PROGRAM LOGPROCESS
VAR_INPUT
	spLogEvent	: STRING;
	spLogComp	: STRING;
	spLogAction	: STRING;
	spLogStatus	: STRING;
	plogFlag		: BOOL;
END_VAR
VAR_OUTPUT
	plog_complete : BOOL := FALSE;
	plog_error	 : BOOL := FALSE;
END_VAR
VAR
	fb_TimeStamp : FB_UpdateTimeStamp ();
	fbCreateDir	 : FB_CreateDir;
	fbFileOpen	 : FB_FileOpen;
	fbFileWrite	 : FB_FilePuts;
	fbFileClose	 : FB_FileClose;
	plog_state	 : ( INIT, 
					 CREATE_DIR, 
					 FILE_OPEN,
					 WRITE_TITLE,
					 WRITE_LOG, 
					 FILE_CLOSE,
					 CLEAR, 
					 ERROR);
					
	pwritepLog	 : STRING[255];
	pwriteTitle	 : STRING;
	spFolderName	 : STRING;
	spwFolderName	 : STRING;
	spFileName	 : STRING;
	spTextLog	 : STRING;
	spwTextLog	 : STRING;
	plastFileName : STRING;	
	spwLogEvent	: STRING;
	spwLogComp	: STRING;
	spwLogAction	: STRING;
	spwLogStatus	: STRING;
	
END_VAR

IF spLogComp<>spwLogComp OR spLogAction<>spwLogAction OR spLogStatus<>spwLogStatus THEN
//	spwLogEvent		:= spLogEvent;
	spwLogComp		:= spLogComp;
	spwLogAction	:= spLogAction;
	spwLogStatus	:= spLogStatus;
ELSE
	RETURN;
END_IF

spTextLog := str_concat(spwLogComp,spwLogAction,spwLogStatus);

WHILE plogFlag DO
	CASE plog_state OF
		// INIT -------------------------------------------------------------------
		INIT:
			plog_complete	:= FALSE;
			plog_error		:= FALSE;
			plog_state 		:= CREATE_DIR;
			fbCreateDir(bExecute:= FALSE);
	
		// CREATE_DIR -------------------------------------------------------------			
		CREATE_DIR:	
			spFolderName := CONCAT('C:\Users\Administrator\Desktop\log\PROCESS\', MAIN.fb_TimeStamp.SystemDate);
//			spFolderName := CONCAT('C:\Users\celli\OneDrive\Desktop\YISB_LOG\PROCESS\', MAIN.fb_TimeStamp.SystemDate);

			IF spFolderName = spwFolderName THEN
				plog_state := FILE_OPEN;
				fbCreateDir(bExecute := FALSE);
				fbFileOpen(bExecute := FALSE);
			ELSE
				fbCreateDir( sPathName:= spFolderName, bExecute:= TRUE );
				IF NOT fbCreateDir.bBusy THEN
					plog_state := FILE_OPEN;
					fbCreateDir(bExecute := FALSE);
					fbFileOpen(bExecute := FALSE);
					spwFolderName := spFolderName;
				END_IF
			END_IF
			
		// FILE_OPEN -------------------------------------------------------------
		FILE_OPEN:
			spFileName := CONCAT(spFolderName,'\');
			spFileName := CONCAT(spFileName, MAIN.fb_TimeStamp.SystemHour);
			spFileName := CONCAT(spFileName,'.csv');
				
			fbFileOpen( sPathName:= spFileName, 
						nMode:= FOPEN_MODEAPPEND, 
						bExecute:= TRUE, 
						hFile=>);
			IF fbFileOpen.bError THEN
				plog_state := ERROR;
				fbFileOpen(bExecute := FALSE);
				fbFileWrite(bExecute := FALSE);
			ELSIF NOT fbFileOpen.bBusy THEN
				plog_state := WRITE_TITLE;
				fbFileOpen(bExecute := FALSE);
				fbFileWrite(bExecute := FALSE);
			END_IF
			
		// WRITE_TITLE -------------------------------------------------------------
		WRITE_TITLE:
			IF plastFileName <> spFileName THEN	
				pwriteTitle := CONCAT('$n','Time Stamp');
				pwriteTitle := CONCAT(pwriteTitle,';');
				pwriteTitle := CONCAT(pwriteTitle,'Component');
				pwriteTitle := CONCAT(pwriteTitle,';');
				pwriteTitle := CONCAT(pwriteTitle,'Action');
				pwriteTitle := CONCAT(pwriteTitle,';');
				pwriteTitle := CONCAT(pwriteTitle,'Status');
				
				fbFileWrite ( hFile:=fbFileOpen.hFile,
								sLine:=pwriteTitle,
								bExecute:=TRUE);
				IF fbFileWrite.bError THEN
					plog_state := ERROR;
					fbFileWrite(bExecute := FALSE);
					fbFileClose(bExecute := FALSE);
				ELSIF NOT fbFileWrite.bBusy THEN
					plog_state := WRITE_LOG;
					fbFileWrite(bExecute := FALSE);
					fbFileClose(bExecute := FALSE);
					plastFileName := spFileName;
				END_IF
			ELSE
				plog_state := WRITE_LOG;
			END_IF

		// WRITE_LOG -------------------------------------------------------------
		WRITE_LOG:	
			pwritepLog := spTextLog;
			
			fbFileWrite ( hFile:=fbFileOpen.hFile,
							sLine:=pwritepLog,
							bExecute:=TRUE);
			IF fbFileWrite.bError THEN
				plog_state := ERROR;
				fbFileWrite(bExecute := FALSE);
				fbFileClose(bExecute := FALSE);
			ELSIF NOT fbFileWrite.bBusy THEN
				plog_state := FILE_CLOSE;
				fbFileWrite(bExecute := FALSE);
				fbFileClose(bExecute := FALSE);
			END_IF
			
		// FILE_CLOSE -------------------------------------------------------------
		FILE_CLOSE:			
			fbFileClose( hFile:=fbFileOpen.hFile,
						 bExecute:=TRUE);
			IF fbFileClose.bError THEN
				plog_state := ERROR;
				fbFileClose(bExecute := FALSE);
			ELSIF NOT fbFileClose.bBusy THEN
				plog_state := CLEAR;
				fbFileClose(bExecute := FALSE);
			END_IF
			
		// CLEAR -------------------------------------------------------------	
		CLEAR:
			plog_complete	:= TRUE;
			plogFlag		:= FALSE;
			plog_state 		:= INIT;
				
		// ERROR -------------------------------------------------------------	
		ERROR:
			plog_error		:= TRUE;
			plogFlag		:= FALSE;
			plog_state 		:= INIT;
	END_CASE
END_WHILE

METHOD str_concat : STRING
VAR_INPUT
	text1	: STRING;
	text2	: STRING;
	text3	: STRING;
END_VAR
VAR
	Con_String : String;
END_VAR
Con_String := CONCAT('$n', MAIN.fb_TimeStamp.FullSystemTime);
Con_String := CONCAT(Con_String, ' ; ');
Con_String := CONCAT(Con_String, text1);
Con_String := CONCAT(Con_String, ' ; ');
Con_String := CONCAT(Con_String, text2);
Con_String := CONCAT(Con_String, ' ; ');
Con_String := CONCAT(Con_String, text3);

str_concat := Con_String;
END_METHOD

END_PROGRAM

(* stored: Version 1.1.0.1, ProductVersion 3.1.4024.12
   POU LOGPROCESS: Id {22f5787e-8e16-45ab-bb8c-d41b9eca7ff5}, SpecialFunc None
   Method str_concat: Id {e94d434c-09ac-414a-9d91-a0fda7e24031} *)
